INTERFACE I_Enumerable EXTENDS __SYSTEM.IQueryInterface

METHOD PUBLIC GetEnumerator : I_ForwardEnumerator
END_METHOD

END_INTERFACE

(* stored: Version 1.1.0.1, ProductVersion 3.1.4024.12
   Itf I_Enumerable: Id {578ac87d-034f-00fe-2fe8-f1abc2d36b90}
   Method GetEnumerator: Id {80dbf027-08b5-0d63-3a9b-4fdf534082d4} *)
